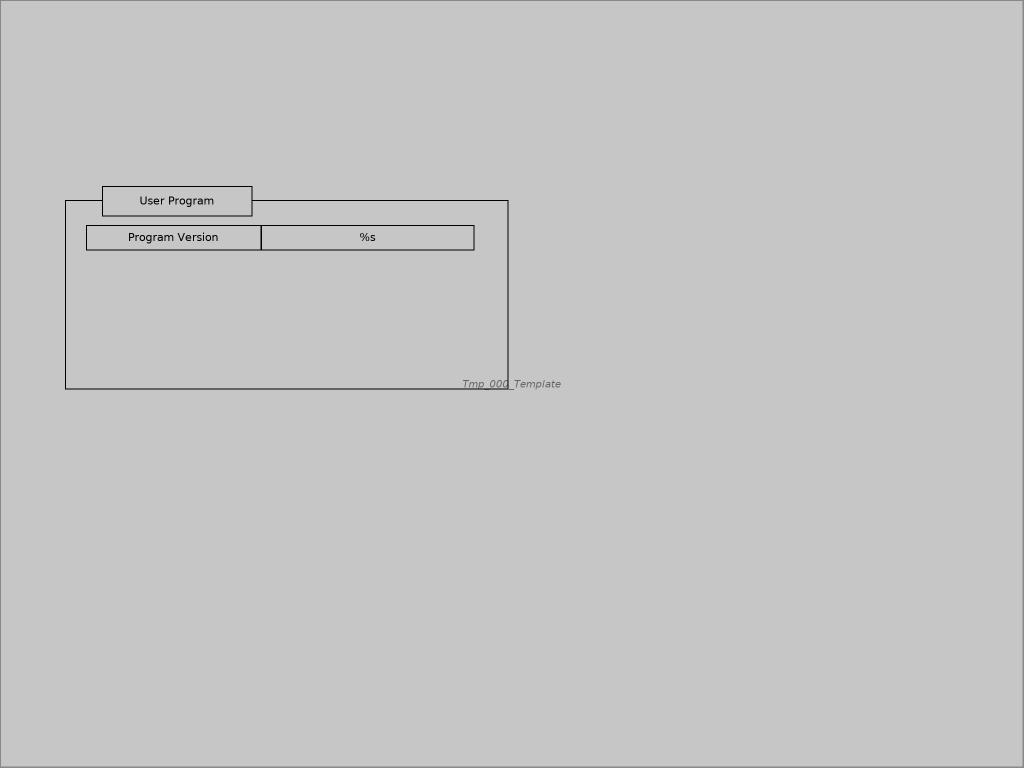
VISUALIZATION Sys_902_Version  // 1024x768
    Frame (0,0 1024x768)
        shows Tmp_000_Template(header := gHMIData.hmiHeader)
    Rectangle (65,200 443x189)
    Rectangle (261,225 213x25), "%s", text variable: stLibVersion_Project_Title.sVersion, text list: ''
    Rectangle (86,225 175x25), "Program Version"
    Rectangle (102,186 150x30), "User Program"
END_VISUALIZATION

(* stored: Version 1.1.0.1, ProductVersion 3.1.4024.11
   Visu Sys_902_Version: Id {871a583d-4806-0ffa-22f6-6f7e0474fa0d} *)
